FUNCTION_BLOCK PearlingHdl

(*
	Description 	: Function bloc to handle pearling unit
	Author		: DLA
	Date		: 09.06.2014
	Version		: 1.00

	Modifications :
                                                                                                                                                                                 
*)

VAR_INPUT
	bEnable									: BOOL;										// Not used
	bPowerOn								: BOOL;										// Power activate
	eCommand								: TModuleCommands;							// Module commande
	bHomeX									: BOOL;										// Axe X Sensor home
	bLimitPosX								: BOOL;										// Axe X Sensor positif limite position
	bLimitNegX								: BOOL;										// Axe X Sensor negatif limite position
	bHomeY									: BOOL;										// Axe Y Sensor home
	bLimitPosY								: BOOL;										// Axe Y Sensor positif limite position 
	bLimitNegY								: BOOL;										// Axe Y Sensor negatif limite position 
	bHomeZ1									: BOOL;										// Axe Z1 Sensor home
	bLimitPosZ1								: BOOL;										// Axe Z1 Sensor positif limite position
	bLimitNegZ1								: BOOL;										// Axe Z1 Sensor negatif limite position
	bHomeZ2									: BOOL;										// Axe Z2 Sensor home
	bLimitPosZ2								: BOOL;										// Axe Z2 Sensor positif limite position
	bLimitNegZ2								: BOOL;										// Axe Z2 Sensor negatif limite position
	bChuck1Opened							: BOOL;										// Chuck Z1 is opened
	bChuck1Closed							: BOOL;										// Chuck Z1 is closed
	bChuck2Opened							: BOOL;										// Chuck Z2 is opened
	bChuck2Closed							: BOOL;										// Chuck Z2 is closed
	bResetErrors							: BOOL;										// Reseting the errors on the module
	bNewJob									: BOOL;										// New job loaded
	bStopReq								: BOOL;										// Request for stoping the module
	bPauseReq								: BOOL;										// Request for pausing the module
	asStickData								: ARRAY[0..1] OF TStickData;				// Description of the sticks used
	asStickDataMMI							: ARRAY[0..1] OF TStickDataMMI;				// Information for the use of the sticks from HMI
	sStickDataShared						: TStickDataShared;							// Information shared betweeen modules for the use of the sticks from HMI
	lrCompenseWeight1						: LREAL;									// Z1 weight compensation
	lrCompenseWeight2						: LREAL;									// Z2 weight compensation
	iComPort								: INT;										// 
	sInTakeFromBarrel						:TGiver;
	iContact1Distance						: INT;
	iContact2Distance						: INT;
	iLoadSensorValue						: INT;
	eSharpenRunStatus						: TRunStatus;
	eBarrelRunStatus						: TRunStatus;
	eRunCommand								: TRunCmdPearling;
	bKeepBothHeadWarm						: BOOL;
	eTableSideForLoader						: TTableSide;
	sPartData								: TPartDataMMI;
	bHead1IsUsed							: BOOL;
	bHead2IsUsed							: BOOL;
	bParallelProduction						: BOOL;
	iLeftVacuumFlow							: INT;
	iRightVacuumFlow						: INT;
	iMachineWO								: DINT;
	iMachineSN								: INT;
	yModulePosition							: BYTE;
END_VAR
VAR_OUTPUT
	bModuleError							: BOOL;
	bXAxisError								: BOOL;
	bYAxisError								: BOOL;
	bZ1AxisError							: BOOL;
	bZ2AxisError							: BOOL;
	bChuck1Error							: BOOL;
	bChuck2Error							: BOOL;
	bSpindle1Error							: BOOL;
	bSpindle2Error							: BOOL;
	bSecurityError							: BOOL;
	bSecurityErrorDetected					: BOOL;
	bMCRError								: BOOL;
	bStick1Broken							: BOOL;
	bStick2Broken							: BOOL;
	bStartPearlingMotor1					: BOOL;
	bStartPearlingMotor2					: BOOL;
	bOpenChuck1								: BOOL;
	bOpenChuck2								: BOOL;
	bActivateEject1							: BOOL;
	bActivateEject2							: BOOL;
	bActivateBlowing1						: BOOL;
	bActivateBlowing2						: BOOL;
	bAspirationPearling1On					: BOOL;
	bAspirationPearling2On					: BOOL;
	bAspirationSharpenOn					: BOOL;
	bStickContact1							: BOOL;
	bStickContact2							: BOOL;
	bCurrent1ReadError						: BOOL;
	bCurrent2ReadError						: BOOL;
	bMotor1Error							: BOOL;
	bMotor2Error							: BOOL;
	bPearlingWeight1OutOfToleranceError		: BOOL;
	bPearlingWeight2OutOfToleranceError		: BOOL;
	bStickNotTakenError						: BOOL;
	bReady2ChangeTool						: BOOL;
	iStickHead								: INT;
	sOutTakeFromBarrel						: TTaker;
	eSharpenRunCmd							: TRunCmdSharpen;
	eBarrelRunCmd							: TRunCmdBarrel;
	eRunStatus								: TRunStatus;
	bManInterlockOut						: BOOL;
	adwMotorRunningHours					: ARRAY[0..1] OF DWORD;
	adwSpindleRunningHours					: ARRAY[0..1] OF DWORD;
	bLeftSpindleUsedWarning					: BOOL;
	bRightSpindleUsedWarning				: BOOL;
	bLeftMotorUsedWarning					: BOOL;
	bRightMotorUsedWarning					: BOOL;
	bLeftSpindleLimitWarning				: BOOL;
	bRightSpindleLimitWarning				: BOOL;
	bLeftSpindleHeatWarning					: BOOL;
	bRightSpindleHeatWarning				: BOOL;
END_VAR
VAR_IN_OUT
	sCurrentState							: TModuleData;
	TManualCmd								: TManPearling;
	sRecData								: ComBuffer;
	sTransData								: ComBuffer;
	asPearlData								: ARRAY[0..1] OF TMMIPearlData;
	sXAxisRef								: AXIS_REF;
	sYAxisRef								: AXIS_REF;
	sZ1AxisRef								: AXIS_REF;
	sZ2AxisRef								: AXIS_REF;
	sRunData								: TRunDataPearling;
	asProbingLog							: ARRAY[0..1] OF  TProbingLog;
END_VAR
VAR PERSISTENT
	alrHighDynParams						: ARRAY[0..3] OF TDynAxisParam;
	alrLowDynParams							: ARRAY[0..3] OF TDynAxisParam;
	alrSafePos								: ARRAY[0..3] OF LREAL;
	alrRobotPos								: ARRAY[0..3,0..PTP_END] OF LREAL;					(* XYZ1Z2 for Ref/Inner/Outer/Drop/... *)
	alrJogStep								: ARRAY[0..3] OF LREAL;								(* Jog step for X,Y,Z1,Z2 *)
	lrSharpeningDelta						: LREAL								:= 10;
	lrSharpenPosOffset						: LREAL								:= 2;
	alrChuckRetractOffset					: ARRAY[0..1] OF LREAL				:= [1,1];		// TODO: HFO, modifier valeur, original [2, 2]
	lrStickTakeSpeed						: LREAL								:= 10;
	bBypassMCR								: BOOL;
(*	iMaxNbOfFwBwSharpen						: INT	:= 1;*)
	TBreakStickDetectTime					: TIME	:= t#30ms;
	aiContactThresholdArea					: ARRAY[0..1, 0..PA_END] OF INT;
	aiSpindleManualSpeed					: ARRAY[0..1] OF INT;
	alrSensorRate							: ARRAY[0..1] OF LREAL								(* in Unit / mm *);
	lrSensorZSpeed							: LREAL								:= 0.1;
	alrLoadSensorOffset						: ARRAY[0..1] OF LREAL;
	lrLoadSensorRate						: LREAL								:= 6.36121;			(* in Unit / g *)
	iLoadSensorTare							: INT								:= 3175;		(* in Unit / g *)
	alrRatiog2mm							: ARRAY[0..1] OF LREAL				:= [2(0.001)];
	lrStickErrorDeltaPos					: LREAL								:= 0.5;
(*	lrSpindelOffsetX						: LREAL								:= 50.0;*)
	iMCROffsetCurrent						: ARRAY[0..1] OF INT				:= [0,0];
	iMCRCurrentRatio						: ARRAY[0..1] OF INT				:= [1,1];
	aiMotorStartedTimeout					: ARRAY[0..1] OF INT 				:= [2000,2000]; (* in ms *)
	aiMotorStoppedTimeout					: ARRAY[0..1] OF INT 				:= [2000,2000]; (* in ms *)
	bForceProbing							: BOOL;
	lrStickOutAfterChange					: LREAL 							:= 12; 			(* mm *)
	lrProbingThreshold						: LREAL								:= 0.05; 		(* mm *)
	alrSharpenTeachZOffset					: LREAL								:= 0.4;
	dwMaxSpindleRunningHours				: DWORD								:= 900;			(*Hours : Max time running spindle before changing it *)
	dwMaxMotorRunningHours					: DWORD								:= 2000;		(*Hours : Max time running motor before changing it *)
	iMCRMinThCurrent						: INT								:= 200;
	iMCRMaxThCurrent 						: INT								:= 800;
	iMCRWarnThCurrent 						: INT								:= 600;
	adwPearlsCounter 						: ARRAY[0..1] OF DWORD				:= [2(0)];
	lrCenterSharpningOffset 				: LREAL 							:= 1.5;
	lrSecurityPreRefPosZ					: LREAL 							:= 1.5;
END_VAR
VAR CONSTANT
	lrLoadSensorStep						: LREAL								:= 0.02;
	lrWeightCalibrationStartOffsetZ			: LREAL 							:= 0.1;
	lrSafeTolerance 						: LREAL 							:= 1;			(* Tolerance for safety Z axis down *)
	lrMaxXYMoveAllowed						: LREAL 							:= 30;			(* Max move authorized when Z axis is down *)
	lrManMaxXYMoveAllowed					: LREAL 							:= 2.1;			(* Max move in manual mode authorized when Z axis is down *)
	lrSecurityRadius						: LREAL								:= 18;
	bInvertX								: BOOL 								:= FALSE;
	bInvertY								: BOOL 								:= FALSE;
	bInvertZ								: BOOL 								:= TRUE;
	lrLayeringCenterOffsetXTable			: LREAL 							:= 65;
	lrLayeringCenterOffsetYTable			: LREAL 							:= 18;
	iHeatOnSpeed							: INT								:= 1000;
END_VAR
VAR
	alrMaxRobotSpeed						: ARRAY[0..3] OF LREAL;
	alrManualRobotSpeed						: ARRAY[0..3] OF LREAL;
	i										: INT;
	j										: INT;
	iAxis									: INT;
	iCurrentManAxis							: INT;
	eRobotXYStatus							: TAxisState;
	aeMoveRobotCommand						: ARRAY[0..3] OF TAxisCommands		:= [4(AC_None)];
	aTRobotAxis								: ARRAY[0..3] OF StdAxis;
	alrCurrentSpeed							: ARRAY[0..3] OF LREAL;
	alrTargetPos							: ARRAY[0..3] OF LREAL;
(*	abForceNewPosZ							: ARRAY[0..1] OF BOOL;*)
	nPearlIndex								: UINT;
	aTPearlingTimer							: ARRAY[0..1] OF TON;
	TCheckTimer								: TON;
	alrPreRefPosZ							: ARRAY[0..1] OF LREAL;
(*	bRemoveXLimitSecurity					: BOOL;
	bRemoveYLimitSecurity					: BOOL;*)
	bManualZIsSafe							: BOOL;
	abChangeStick							: ARRAY[0..1] OF BOOL				:= [TRUE,TRUE];
	abSharpenStick							: ARRAY[0..1] OF BOOL				:= [TRUE,TRUE];
	abDoProbing								: ARRAY[0..1] OF BOOL;
	abRetryProbing							: ARRAY[0..1] OF BOOL;
	abProbingDone							: ARRAY[0..1] OF BOOL;
	aiProbingCount							: ARRAY[0..1] OF INT;
	alrProbingStartPos						: ARRAY[0..1] OF LREAL;
	eStickStep								: TModuleSteps;
	aeProbingStep							: ARRAY[0..1] OF TModuleSteps;
	TCheckTime								: TIME								:= T#5S;
	TMCRDrv									: MCRDrv;
	aTCheckChuck							: ARRAY[0..1] OF FB_CheckJack1_2;
	alrCorrectionMCR						: ARRAY[0..1] OF LREAL;
	eMCRCommand								: TMCRCommands;
	bMCRReady								: BOOL;
(*	abLastStickContact						: ARRAY[0..1] OF BOOL;*)
	aiNbOfPearlsDone						: ARRAY[0..1] OF INT;
	iCurrentArea							: INT;
	aArea									: ARRAY[0..C_MAX_NB_OF_PEARLS] OF TPearlsArea;
	alrPearlingEnergy						: ARRAY[0..1] OF LREAL;
	aTDispersion							: ARRAY[0..1] OF Dispersion;
	alrRemainingStickLength					: ARRAY[0..1] OF LREAL;
	aTMotorCounter							: ARRAY[0..1] OF RunningCounter;
	aTSpindleCounter						: ARRAY[0..1] OF RunningCounter;
	TWaitChuckOpen							: TON;
	abZRefTaken								: ARRAY[0..3,0..1,0..1] OF BOOL; 					(*Layring , Offset Layring, Head *)
	alrSecurityPosition						: ARRAY[0..3,0..1,0..1] OF LREAL;					(*Layring , Offset Layring, Head *)
	alrContactPosition						: ARRAY[0..3,0..1,0..1] OF LREAL;					(*Layring , Offset Layring, Head *)
	alrContactStickPosition					: ARRAY[0..3,0..1,0..1] OF LREAL;					(*Layring , Offset Layring, Head *)
	alrProbingRef							: ARRAY[0..3,0..1,0..1] OF LREAL; 					(*Layring , Offset Layring, Head *)
	alrHeadSecurityPosition					: ARRAY[0..1] OF LREAL;
	alrHeadContactPosition					: ARRAY[0..1] OF LREAL;
	alrHeadContactStickPosition				: ARRAY[0..1] OF LREAL;
	alrHeadProbingRef						: ARRAY[0..1] OF LREAL;
	alrSharpenProbing						: ARRAY[0..1] OF LREAL;
	alrDeltaSharpenProbing					: ARRAY[0..1] OF LREAL;
	alrStickCorrection						: ARRAY[0..1] OF LREAL;
	alrDeltaStickCorrection					: ARRAY[0..1] OF LREAL;
	alrFirstPearlCorrection					: ARRAY[0..1] OF LREAL;
	abTakeZRef								: ARRAY[0..1] OF BOOL;
	bClearZRef								: BOOL;
	abNeedSharpening						: ARRAY[0..1] OF BOOL;
	abNeedChangeStick						: ARRAY[0..1] OF BOOL;
	bFirstStart								: BOOL								:= TRUE;
	bFirstInit								: BOOL								:= TRUE;
	abBadPearling							: ARRAY[0..1] OF BOOL;
	alrDynParams							: ARRAY[0..3] OF TDynAxisParam;
	yMCRChannel								: BYTE;
	abPearlStarted							: ARRAY[0..1] OF BOOL;
	abPearlDone								: ARRAY[0..1] OF BOOL;
	abPearlPosReached						:  ARRAY[0..1] OF BOOL;
	lrRadius								: LREAL;
	alrLastProbingPos						: ARRAY[0..1] OF LREAL;
	aTWaitMotorStarted						: ARRAY[0..1] OF TON;
	aTWaitMotorStopped						: ARRAY[0..1] OF TON;
	iNbOfFwBwSharpen						: INT;
	iNbOfFwBwSharpenBeforeMove				: INT;
	abNewStick								: ARRAY[0..1] OF BOOL				:= [FALSE,FALSE];
	iDebugPos								: INT;
	iDebugSide								: INT;
	aTDetectStickBroken						: ARRAY[0..1] OF TON;
(*	bZIsSafe								: BOOL;*)
	alrProbingPos							: ARRAY[0..1] OF LREAL;
	alrCheckProbingPos						: ARRAY[0..1] OF LREAL;
	alrProbingLimit							: ARRAY[0..1] OF LREAL;
(*	iNbOfPearlsRemainingOnThisArea			: INT;*)
	abCheckingStick							: ARRAY[0..1] OF BOOL;
	TWaitCurrentMotorBeltOk					: TON;
	TWaitCurrentMotorWarmOk					: TON;
	aTStickContactValidated					: ARRAY[0..1] OF TON;
	TStickContactValidTime					: TIME								:= T#250MS; // valeur original ==> t#500ms; Temps de stabilisation du capteur de de distance en contacte
	TStickStabilisationTime					: TIME								:= T#400MS;	// Temps pour stabiliser le capteur de distance sans contact
	aIMinPos								: ARRAY[0..1] OF INT;
	alrDeltaZPearl							: ARRAY[0..1] OF LREAL;
	alrDeltaWeightPearl						: ARRAY[0..1] OF LREAL;
	iTableIndex								: INT;
	lrBasePos								: LREAL;
(*	TWaitEjectorTimer						: TON;*)
	abWeightTableValid						: ARRAY[0..1] OF BOOL;
	alrWeightTable							: ARRAY[0..1,0..C_WEIGHT_TABLE_MAX] OF LREAL;
	iSide									: INT;
	abStartPearlingMotor					: ARRAY[0..1] OF BOOL;
	aiContactDistance						: ARRAY[0..1] OF INT;
	abUseSpindle							: ARRAY[0..1] OF BOOL;
	abChuckOpened							: ARRAY[0..1] OF BOOL;
	abChuckClosed							: ARRAY[0..1] OF BOOL;
	abOpenChuck								: ARRAY[0..1] OF BOOL;
	abActivateEject							: ARRAY[0..1] OF BOOL;
	abSpindleError							: ARRAY[0..1] OF BOOL;
	abAspirationPearling					: ARRAY[0..1] OF BOOL;
	abStickContact							: ARRAY[0..1] OF BOOL;
	abActivateBlowing						: ARRAY[0..1] OF BOOL;
	abCurrentReadError						: ARRAY[0..1] OF BOOL;
	abMotorError							: ARRAY[0..1] OF BOOL;
	abSpindleCurrentOk						: ARRAY[0..1] OF BOOL;
	abStickBroken							: ARRAY[0..1] OF BOOL;
	abStickBrokenDetected					: ARRAY[0..1] OF BOOL;
	abPearlNeeded							: ARRAY[0..1] OF BOOL;
	abHeadIsUsed							: ARRAY[0..1] OF BOOL;
	abPearlingWeightOutOfToleranceError		: ARRAY[0..1] OF BOOL;
	abPearlingWeightOutOfToleranceDetected	: ARRAY[0..1] OF BOOL;
	abFirstPearl							: ARRAY[0..1] OF BOOL;
	aiCountPearlError						: ARRAY[0..1] OF INT;
	alrBasePearlingEnergy					: ARRAY[0..1] OF LREAL;
	alrCompenseWeight						: ARRAY[0..1] OF LREAL;
	aiPearlingLayringPos					: ARRAY[0..1] OF INT;
	aiPearlingLayringOffsetPos				: ARRAY[0..1] OF INT;
	anPearlIndexDone						: ARRAY[0..1] OF UINT;
	aiSideInfo								: ARRAY[0..1] OF INT;
	TLayeringCenter							:  TPositionXY;
	TPearlPosition							:  TPositionXY;
	iFirstHeadUsed							: INT;
	iRejectPos								: INT;
	iChangeStickPos							: INT;
	nPearl									: UINT;
	aiPearlingTeachedPos					: ARRAY[0..1] OF INT;
	alrPearlingOffset						: ARRAY[0..4] OF LREAL;
	alrPearlingInvert						: ARRAY[0..4] OF LREAL;
	alrHeadPushed_mm						: ARRAY[0..1] OF LREAL;
(*	psPartData								: ARRAY[0..1] OF POINTER TO TPartData;*)
	bChangeToolSide							: BOOL;
(*	bChangeTool								: BOOL;*)
	bEndPearling							: BOOL;
	lrWeight								: LREAL;
	lrMaxMCRCorrection						: LREAL;
	bCalibrationInProgress					: BOOL;
	aeProbingArea							: ARRAY[0..1] OF TProbingArea;
	TDebug									: TPearlingDebug;
	aePearlingArea							: ARRAY[0..1] OF TProbingArea;
	TWaitHeadStab							: TON;
	atStickValidateTime						: ARRAY[0..1] OF LREAL;
	aiVacuumFlow							: ARRAY[0..1] OF INT;
	ayChannelStatus							: ARRAY[0..1] OF BYTE;
	abCurrentLimitWarning					: ARRAY[0..1] OF BOOL;
	aTWaitSpindleHeatOn						: ARRAY[0..1] OF TON;
	aTDetectSpindleCooled					: ARRAY[0..1] OF TON;
	abNeedSpindleHeatOn						: ARRAY[0..1] OF BOOL;
	ai_ProbingStep							: ARRAY [0..1] OF INT;
	i_StickStep								: INT;
	iDebugPosBrokenStick					: INT;
END_VAR


(*_AppInfo.BootDataLoaded;			// HFO, to know if boot data was loaded
_AppInfo.OldBootData;
_AppInfo.PersistentStatus;*)

(* Optimize code *)
abStartPearlingMotor[PH_Left] := bStartPearlingMotor1;
abStartPearlingMotor[PH_Right] := bStartPearlingMotor2;
aiContactDistance[PH_Left] := iContact1Distance;
aiContactDistance[PH_Right] := iContact2Distance;
abChuckOpened[PH_Left] := bChuck1Opened;
abChuckOpened[PH_Right] := bChuck2Opened;
abChuckClosed[PH_Left] := bChuck1Closed;
abChuckClosed[PH_Right] := bChuck2Closed;
alrCompenseWeight[PH_Left] := lrCompenseWeight1;
alrCompenseWeight[PH_Right] := lrCompenseWeight2;
abHeadIsUsed[PH_Left] := bHead1IsUsed;
abHeadIsUsed[PH_Right] := bHead2IsUsed;
aiVacuumFlow[PH_LEFT] := iLeftVacuumFlow;
aiVacuumFlow[PH_RIGHT] := iRightVacuumFlow;

eSharpenRunCmd := RCS_None;
eBarrelRunCmd := RCB_None;

IF bInvertX THEN
	alrPearlingInvert[PA_X] := -1;
ELSE
	alrPearlingInvert[PA_X] := 1;
END_IF
IF bInvertY THEN
	alrPearlingInvert[PA_Y] := -1;
ELSE
	alrPearlingInvert[PA_Y] := 1;
END_IF
IF bInvertZ THEN
	alrPearlingInvert[PA_Z1] := -1;
	alrPearlingInvert[PA_Z2] := -1;
ELSE
	alrPearlingInvert[PA_Z1] := 1;
	alrPearlingInvert[PA_Z2] := 1;
END_IF

FOR iAxis := 0 TO 3 DO
	alrMaxRobotSpeed[iAxis] := aTRobotAxis[iAxis].lrRunningSpeed;
	alrManualRobotSpeed[iAxis] := aTRobotAxis[iAxis].lrManualSpeed;
END_FOR

IF (NOT sCurrentState.bStepMode) THEN
	sCurrentState.bWaitStep := FALSE;
END_IF

IF bFirstStart THEN
	FOR iSide := 0 TO 1 DO
		abWeightTableValid[iSide] := FALSE;
		aTDetectSpindleCooled[iSide](IN := FALSE);
		aTWaitSpindleHeatOn[iSide](IN := FALSE);
		abNeedSpindleHeatOn[iSide] := TRUE;
	END_FOR
	bFirstStart := FALSE;
END_IF

IF bNewJob THEN
	FOR iSide := 0 TO 1 DO
		abSharpenStick[iSide] := TRUE;
		aiNbOfPearlsDone[iSide] := 1;
	END_FOR
	bClearZRef := TRUE;
END_IF

FOR iSide:=0 TO 1 DO
	abStickContact[iSide] := aiContactDistance[iSide] > (aiContactThresholdArea[iSide , aeProbingArea[iSide]] + 0.05 * alrSensorRate[iSide]);
	aTWaitMotorStarted[iSide](IN := abStartPearlingMotor[iSide],PT := INT_TO_TIME(aiMotorStartedTimeout[iSide]));
	aTWaitMotorStopped[iSide](IN := NOT abStartPearlingMotor[iSide],PT := INT_TO_TIME(aiMotorStoppedTimeout[iSide]));
	aTMotorCounter[iSide](bStart := abStartPearlingMotor[iSide], bReset := FALSE);
	aTSpindleCounter[iSide](bStart := abStartPearlingMotor[iSide], bReset := FALSE);
	IF NOT abDoProbing[iSide] THEN
		abProbingDone[iSide] := FALSE;
	END_IF
	(* For debug purpose *)
	IF alrSensorRate[iSide] <> 0 THEN
		alrHeadPushed_mm[iSide] := INT_TO_REAL(LREAL_TO_INT(((aiContactDistance[iSide]-aiContactThresholdArea[iSide , aeProbingArea[iSide]])/alrSensorRate[iSide])*100))/100.0;
	ELSE
		alrHeadPushed_mm[iSide] := 0;
	END_IF
	alrBasePearlingEnergy[iSide] := sRunData.sPearlingData.iWeight +  alrCompenseWeight[iSide];
	IF bParallelProduction THEN
		aiSideInfo[iSide] := 0;
	ELSE
		aiSideInfo[iSide] := iSide;
	END_IF
END_FOR

(* For debug purpose *)
IF lrLoadSensorRate<>0 THEN
	lrWeight := (INT_TO_LREAL(iLoadSensorValue) - INT_TO_LREAL(iLoadSensorTare)) / lrLoadSensorRate;
ELSE
	lrWeight := 0;
END_IF

CASE eCommand OF
	MC_NoCmd :
		CASE sCurrentState.eStatus OF
			MS_Init :
				CASE sCurrentState.eStep OF
(*----------------- Init ------------------*)
					SP_InitStp1 :
						FOR iSide := 0 TO 1 DO
							abAspirationPearling[iSide] := FALSE;
							abActivateEject[iSide] := FALSE;
							(* Move Z Up *)
							aeMoveRobotCommand[PA_Z1+iSide] := AC_MoveLimitNeg;
						END_FOR
						bAspirationSharpenOn := FALSE;
						alrCurrentSpeed := alrMaxRobotSpeed;
						sCurrentState.eStep := SP_InitStp2;
					SP_InitStp2 :
						IF aTRobotAxis[PA_Z1].eCurrentState = AS_OnLimitNeg  AND
						     aTRobotAxis[PA_Z2].eCurrentState = AS_OnLimitNeg THEN
							(* Init X / Y*)
							aeMoveRobotCommand[PA_X] := AC_Init;
							aeMoveRobotCommand[PA_Y] := AC_Init;
							sCurrentState.eStep := SP_InitStp3;
						END_IF
					SP_InitStp3 :
						IF 	(aTRobotAxis[PA_X].eCurrentState = AS_InPosition) AND
							(aTRobotAxis[PA_Y].eCurrentState = AS_InPosition) THEN
							(* Move X/ Y to Safe *)
							alrTargetPos[PA_X] := alrSafePos[PA_X];
							alrTargetPos[PA_Y] := alrSafePos[LA_Y];
							aeMoveRobotCommand[PA_X] := AC_MoveAtAbsPos;
							aeMoveRobotCommand[PA_Y] := AC_MoveAtAbsPos;
							sCurrentState.eStep := SP_InitStp4;
						END_IF
					SP_InitStp4 :
						IF aTRobotAxis[PA_X].eCurrentState = AS_InPosition AND
						     aTRobotAxis[PA_Y].eCurrentState = AS_InPosition THEN
								(* Init Z *)
								aeMoveRobotCommand[PA_Z1] := AC_Init;
								aeMoveRobotCommand[PA_Z2] := AC_Init;
								sCurrentState.eStep := SP_InitStp5;
						END_IF
					SP_InitStp5 :
						IF aTRobotAxis[PA_Z1].eCurrentState=AS_InPosition AND
							aTRobotAxis[PA_Z2].eCurrentState=AS_InPosition THEN
							(* Move Z to Safe *)
							alrTargetPos[PA_Z1] := alrSafePos[PA_Z1];
							alrTargetPos[PA_Z2] := alrSafePos[LA_Z2];
							aeMoveRobotCommand[PA_Z1] := AC_MoveAtAbsPos;
							aeMoveRobotCommand[PA_Z2] := AC_MoveAtAbsPos;
							sCurrentState.eStep := SP_InitStp6;
						END_IF
					SP_InitStp6 :
						IF  aTRobotAxis[PA_Z1].eCurrentState = AS_InPosition AND
						     aTRobotAxis[PA_Z2].eCurrentState = AS_InPosition THEN
							IF bBypassMCR THEN
								sCurrentState.eStep := SP_InitStp99;
							ELSIF bMCRReady THEN
								yMCRChannel := 1;
								sCurrentState.eStep := SP_InitStp10;
							END_IF
						END_IF
					SP_InitStp10 :
						(* Configure MCR *)
						eMCRCommand := MCRC_ConfigMeasure;
						sCurrentState.eStep := SP_InitStp11;
					SP_InitStp11 :
						IF bMCRReady THEN
							IF yMCRChannel = 1 THEN
								yMCRChannel := 2;
								sCurrentState.eStep := SP_InitStp10;
							ELSE
								yMCRChannel := 1;
								sCurrentState.eStep := SP_InitStp12;
							END_IF
						END_IF
					SP_InitStp12 :
						eMCRCommand := MCRC_SetRatio;
						TMCRDrv.lrRatio := asStickDataMMI[yMCRChannel - 1].lrMCRRatio;
						sCurrentState.eStep := SP_InitStp13;
					SP_InitStp13 :
						IF bMCRReady THEN
							IF yMCRChannel = 1 THEN
								yMCRChannel := 2;
								sCurrentState.eStep := SP_InitStp12;
							ELSE
								yMCRChannel := 1;
								sCurrentState.eStep := SP_InitStp14;
							END_IF
						END_IF
					SP_InitStp14 :
						(* Do spindle heat on if needed *)
						TMCRDrv.iSpeedSetpoint := iHeatOnSpeed;;
						eMCRCommand := MCRC_SetSpeed;
						sCurrentState.eStep := SP_InitStp15;
					SP_InitStp15 :
						IF bMCRReady THEN
							IF yMCRChannel = 1 THEN
								yMCRChannel := 2;
								sCurrentState.eStep := SP_InitStp14;
							ELSE
								yMCRChannel := 1;
								sCurrentState.eStep := SP_InitStp16;
							END_IF
						END_IF
					SP_InitStp16 :
						abStartPearlingMotor[PH_Left] := abNeedSpindleHeatOn[PH_Left];
						abStartPearlingMotor[PH_Right] := abNeedSpindleHeatOn[PH_Right];
						sCurrentState.eStep := SP_InitStp17;
					SP_InitStp17 :
						IF (NOT (abNeedSpindleHeatOn[PH_Left] AND abStartPearlingMotor[PH_Left]) AND 
								NOT (abNeedSpindleHeatOn[PH_Right] AND abStartPearlingMotor[PH_Right])) THEN
							sCurrentState.eStep := SP_InitStp25;
						END_IF
					SP_InitStp25 :
						eMCRCommand := MCRC_SetSpeed;
						TMCRDrv.iSpeedSetpoint := sStickDataShared.sStickDataMMIShared.iMCRSharpenSpeed;
						sCurrentState.eStep := SP_InitStp26;
					SP_InitStp26 :
						IF bMCRReady THEN
							IF yMCRChannel = 1 THEN
								yMCRChannel := 2;
								sCurrentState.eStep := SP_InitStp25;
							ELSE
								yMCRChannel := 1;
								sCurrentState.eStep := SP_InitStp27;
							END_IF
						END_IF
					SP_InitStp27:
						(* Set Parameter*)
						IF NOT bFirstInit THEN
							eMCRCommand := MCRC_SetParam;
							TMCRDrv.iOffsetCurrent := iMCROffsetCurrent[yMCRChannel - 1];
							TMCRDrv.iCurrentRatio := iMCRCurrentRatio[yMCRChannel - 1];
						END_IF
						sCurrentState.eStep := SP_InitStp28;
					SP_InitStp28:
						IF bMCRReady THEN
							IF yMCRChannel = 1 THEN
								yMCRChannel := 2;
								sCurrentState.eStep := SP_InitStp27;
							ELSE
								yMCRChannel := 1;
								sCurrentState.eStep := SP_InitStp29;
							END_IF
						END_IF
					SP_InitStp29:
						(* Set threshold*)
						eMCRCommand := MCRC_DefineCurrentThr;
						TMCRDrv.iMinThCurrent := iMCRMinThCurrent;
						TMCRDrv.iMaxThCurrent := iMCRMaxThCurrent;
						TMCRDrv.iWarnThCurrent := iMCRWarnThCurrent;
						sCurrentState.eStep := SP_InitStp30;
					SP_InitStp30:
						IF bMCRReady THEN
							IF yMCRChannel = 1 THEN
								yMCRChannel := 2;
								sCurrentState.eStep := SP_InitStp29;
							ELSE
								yMCRChannel := 1;
								sCurrentState.eStep := SP_InitStp31;
							END_IF
						END_IF
					SP_InitStp31:
						IF NOT bFirstInit THEN
							(* Set MachineID*)
							eMCRCommand := MCRC_DefineMachineID;
							TMCRDrv.iMachineWO := iMachineWO;
							TMCRDrv.iMachineSN := iMachineSN;
							TMCRDrv.yMachineSide := asc('a') + yModulePosition;
						END_IF
						sCurrentState.eStep := SP_InitStp32;
					SP_InitStp32:
						IF bMCRReady THEN
							IF yMCRChannel = 1 THEN
								yMCRChannel := 2;
								sCurrentState.eStep := SP_InitStp31;
							ELSE
								yMCRChannel := 1;
								sCurrentState.eStep := SP_InitStp99;
							END_IF
						END_IF
					SP_InitStp50: (*Init if already init done, always move Z to safe *)
						(* Go to safe position *)
						alrCurrentSpeed := alrMaxRobotSpeed;
						alrTargetPos[PA_Z1] := alrSafePos[PA_Z1];
						alrTargetPos[PA_Z2] := alrSafePos[PA_Z2];
						aeMoveRobotCommand[PA_Z1] := AC_MoveAtAbsPos;
						aeMoveRobotCommand[PA_Z2] := AC_MoveAtAbsPos;
						sCurrentState.eStep := SP_InitStp51;
					SP_InitStp51 :
						IF 	(aTRobotAxis[PA_Z1].eCurrentState = AS_InPosition) AND
							(aTRobotAxis[PA_Z2].eCurrentState = AS_InPosition) THEN
							sCurrentState.eStep := SP_InitStp99;
						END_IF
					SP_InitStp99 :
						bFirstInit := FALSE;
						FOR iSide := 0 TO 1 DO
							abDoProbing[iSide] := FALSE;
							abUseSpindle[iSide] := FALSE;
							abRetryProbing[iSide] := FALSE;
							aiProbingCount[iSide] := 0;
						END_FOR
						sCurrentState.eStatus := MS_Ready;
						sCurrentState.bInitDone := TRUE;
						sCurrentState.eStep := SP_RunStp1;
						eStickStep := SP_RunStp1;
						aeProbingStep[PH_Left] := SP_RunStp1;
						aeProbingStep[PH_Right] := SP_RunStp1;

				END_CASE
			MS_Running :
				IF (NOT sCurrentState.bWaitStep) THEN
(*----------------- Probing ------------------*)
					FOR iSide := 0 TO 1 DO
						CASE aeProbingStep[iSide] OF
							SP_RunStp1 :
								IF abDoProbing[iSide] THEN
									aiProbingCount[iSide] := 0;
									alrProbingStartPos[iSide] := alrTargetPos[PA_Z1 + iSide];
									abProbingDone[iSide] := FALSE;
									abStartPearlingMotor[iSide] := FALSE;
									aeProbingStep[iSide] := SP_RunStp20;
								END_IF
							SP_RunStp20:
								(* Continuous move probing with analog sensor *)
								IF (aTRobotAxis[PA_Z1+ iSide].eCurrentState = AS_InPosition) AND aTWaitMotorStopped[iSide].Q THEN
									(* Move 0.5 mm above probing pos to check default sensor value *)
									alrTargetPos[PA_Z1 + iSide] := alrProbingStartPos[iSide] - 0.5;		// TODO : HFO modifier valeur en dure, original 0.5
									alrCurrentSpeed[PA_Z1 + iSide] := alrMaxRobotSpeed[PA_Z1 + iSide];
									aeMoveRobotCommand[PA_Z1 + iSide] := AC_MoveAtAbsPos;
									aTStickContactValidated[iSide](IN := FALSE);
									aeProbingStep[iSide] := SP_RunStp21;
								END_IF
							SP_RunStp21:
								IF (aTRobotAxis[PA_Z1 + iSide].eCurrentState = AS_InPosition) THEN
									aTStickContactValidated[iSide](IN := TRUE,PT := TStickStabilisationTime);	// Valueur original ==> PT := TStickContactValidTime
									IF aTStickContactValidated[iSide].Q THEN
										asProbingLog[iSide].iPreviousProbingThreshold := aiContactThresholdArea[iSide , aeProbingArea[iSide]];
										aiContactThresholdArea[iSide , aeProbingArea[iSide]] := aiContactDistance[iSide];
										(* Move down 0.5mm *)
										alrTargetPos[PA_Z1 + iSide] := alrProbingStartPos[iSide]- 0.3;  		// TODO : HFO, Ajout de valeur negative
										//alrTargetPos[PA_Z1 + iSide] := alrProbingStartPos[iSide];
										aeMoveRobotCommand[PA_Z1 + iSide] := AC_MoveAtAbsPos;
										aTStickContactValidated[iSide](IN := FALSE);
										aeProbingStep[iSide] := SP_RunStp25;
									END_IF
								END_IF
							SP_RunStp25:
								IF (aTRobotAxis[PA_Z1 + iSide].eCurrentState = AS_InPosition) THEN
									aTStickContactValidated[iSide](IN := TRUE,PT := TStickContactValidTime);
									IF aTStickContactValidated[iSide].Q THEN
										(* Check if we must go up or down *)
										IF (aiContactDistance[iSide] > aiContactThresholdArea[iSide , aeProbingArea[iSide]] + alrSensorRate[iSide] * lrProbingThreshold) THEN
											(* Go up *)
											aeProbingStep[iSide] := SP_RunStp30;
										ELSE
											(* Go down *)
											aeProbingStep[iSide] := SP_RunStp40;
										END_IF								
									END_IF
								END_IF	
							SP_RunStp30:
								(* Move up slowly until we get contact *)
								alrTargetPos[PA_Z1 + iSide] := alrProbingStartPos[iSide] - 2;
								alrCurrentSpeed[PA_Z1 + iSide] := lrSensorZSpeed;
								aeMoveRobotCommand[PA_Z1 + iSide] := AC_MoveAtAbsPos;
								aeProbingStep[iSide] := SP_RunStp35;
							SP_RunStp35:
								IF (aiContactDistance[iSide] < aiContactThresholdArea[iSide , aeProbingArea[iSide]] + alrSensorRate[iSide] * lrProbingThreshold) THEN
									aTStickContactValidated[iSide](IN := FALSE);
									aeMoveRobotCommand[PA_Z1 + iSide] := AC_Stop;
									aeProbingStep[iSide] := SP_RunStp50;
									sCurrentState.bWaitStep := TRUE;
								ELSIF (aTRobotAxis[PA_Z1 + iSide].eCurrentState = AS_InPosition) THEN
									aeMoveRobotCommand[PA_Z1] := AC_Stop;
									aeMoveRobotCommand[PA_Z2] := AC_Stop;
									bSecurityError := TRUE;
									iDebugPos := 1;
									iDebugSide := iSide;
								END_IF
							SP_RunStp40:
								(* Move down slowly until we get contact *)
								alrTargetPos[PA_Z1 + iSide] := alrProbingLimit[iSide];
								alrCurrentSpeed[PA_Z1 + iSide] := lrSensorZSpeed;
								aeMoveRobotCommand[PA_Z1 + iSide] := AC_MoveAtAbsPos;
								aeProbingStep[iSide] := SP_RunStp45;
							SP_RunStp45:
								IF (aiContactDistance[iSide] > aiContactThresholdArea[iSide , aeProbingArea[iSide]] + alrSensorRate[iSide] * lrProbingThreshold) THEN
									aTStickContactValidated[iSide](IN := FALSE);
									aeMoveRobotCommand[PA_Z1 + iSide] := AC_Stop;
									aeProbingStep[iSide] := SP_RunStp50;
									sCurrentState.bWaitStep := TRUE;
								ELSIF (aTRobotAxis[PA_Z1 + iSide].eCurrentState = AS_InPosition) THEN
									aeMoveRobotCommand[PA_Z1] := AC_Stop;
									aeMoveRobotCommand[PA_Z2] := AC_Stop;
									bSecurityError := TRUE;
									iDebugPos := 10;
									iDebugSide := iSide;
								END_IF
							SP_RunStp50:
								IF (aTRobotAxis[PA_Z1 + iSide].eCurrentState = AS_InPosition) THEN
									aTStickContactValidated[iSide](IN := TRUE,PT := TStickContactValidTime);
									IF aTStickContactValidated[iSide].Q THEN
										alrProbingPos[iSide] := aTRobotAxis[PA_Z1 + iSide].lrCurrentPos - (aiContactDistance[iSide] - aiContactThresholdArea[iSide , aeProbingArea[iSide]])/alrSensorRate[iSide];
										(* Move 2 mm above probing pos to check 1st measure *)
										alrTargetPos[PA_Z1 + iSide] := aTRobotAxis[PA_Z1 + iSide].lrCurrentPos - 2;
										alrCurrentSpeed[PA_Z1 + iSide] := alrMaxRobotSpeed[PA_Z1 + iSide];
										aeMoveRobotCommand[PA_Z1 + iSide] := AC_MoveAtAbsPos;
										aeProbingStep[iSide] := SP_RunStp55;
									END_IF
								END_IF
							SP_RunStp55:
								IF (aTRobotAxis[PA_Z1 + iSide].eCurrentState = AS_InPosition) AND NOT asProbingLog[iSide].bNewLog THEN
									(* Move to contact position *)
									alrTargetPos[PA_Z1 + iSide] := alrTargetPos[PA_Z1 + iSide]+2;
									aeMoveRobotCommand[PA_Z1 + iSide] := AC_MoveAtAbsPos;
									aTStickContactValidated[iSide](IN := FALSE);
									aeProbingStep[iSide] := SP_RunStp60;
								END_IF
							SP_RunStp60:
								IF (aTRobotAxis[PA_Z1 + iSide].eCurrentState = AS_InPosition) THEN
									aTStickContactValidated[iSide](IN := TRUE,PT := TStickContactValidTime);
									IF aTStickContactValidated[iSide].Q THEN
										alrCheckProbingPos[iSide] := aTRobotAxis[PA_Z1 + iSide].lrCurrentPos - (aiContactDistance[iSide] - aiContactThresholdArea[iSide , aeProbingArea[iSide]])/alrSensorRate[iSide];
										asProbingLog[iSide].alrProbingPos[PH_Left] := alrProbingPos[iSide];
										asProbingLog[iSide].alrProbingPos[PH_Right] := alrCheckProbingPos[iSide];
										asProbingLog[iSide].eProbingArea := aeProbingArea[iSide];
										asProbingLog[iSide].iProbingThreshold := aiContactThresholdArea[iSide , aeProbingArea[iSide]];
										asProbingLog[iSide].bNewLog := TRUE;
(* DLA										IF (ABS(alrProbingPos[iSide] - alrCheckProbingPos[iSide]) < 0.1) THEN *)
										IF (ABS(alrProbingPos[iSide] - alrCheckProbingPos[iSide]) < 0.3) THEN
											abProbingDone[iSide] := TRUE;
											aeProbingStep[iSide] := SP_RunStp70;
										ELSIF abRetryProbing[iSide] AND aiProbingCount[iSide] < 3 AND (ABS(alrProbingPos[iSide] - alrCheckProbingPos[iSide]) < 0.3)THEN
											aiProbingCount[iSide] := aiProbingCount[iSide] + 1;
											aeProbingStep[iSide] := SP_RunStp20;
										ELSE
											bSecurityError := TRUE;
											iDebugPos := 2;
											iDebugSide := iSide;
										END_IF
									END_IF
								END_IF
							SP_RunStp70:
								IF NOT abDoProbing[iSide] THEN
									aeProbingStep[iSide] := SP_RunStp1;
								END_IF
						END_CASE
					END_FOR
(*----------------- Stick gestion ------------------*)
					CASE eStickStep OF
						SP_RunStp1 :
							IF (aTRobotAxis[PA_Z1].eCurrentState = AS_InPosition) AND (aTRobotAxis[PA_Z2].eCurrentState = AS_InPosition) THEN
								FOR iSide := 0 TO 1 DO
									IF abChangeStick[iSide] AND abUseSpindle[iSide] THEN
										abSharpenStick[iSide] := TRUE;
										eStickStep := SP_RunStp2; (* Change Stick [Serial]*)
									END_IF
								END_FOR
								IF (eStickStep <> SP_RunStp2) THEN
									FOR iSide := 0 TO 1 DO
										IF abSharpenStick[iSide] AND abUseSpindle[iSide] THEN
											IF NOT abChuckClosed[iSide] THEN
												abSharpenStick[iSide] := FALSE;
											ELSE
												IF abNewStick[iSide] OR aiNbOfPearlsDone[iSide]>0 THEN
													eStickStep := SP_RunStp50; (* Sharpen [parallel]*)
												ELSIF NOT abNewStick[iSide] AND abSharpenStick[iSide] AND aiNbOfPearlsDone[iSide]=0 THEN
													(* sharpen is not need if no pearl has been made *)
													abSharpenStick[iSide] := FALSE;
												END_IF
											END_IF
										END_IF
									END_FOR
								END_IF
							END_IF
						SP_RunStp2 : (* Change Stick [Serial]*)
							FOR iSide := 0 TO 1 DO
								(* Stop motors *)
								abStartPearlingMotor[iSide] := FALSE;
								(* Move Z to safe *)
								alrTargetPos[PA_Z1+iSide] := alrSafePos[PA_Z1+iSide];
								aeMoveRobotCommand[PA_Z1+iSide] := AC_MoveAtAbsPos;
							END_FOR
							eStickStep := SP_RunStp10;
						SP_RunStp10 :  (* Reject Stick [Serial]*)
							IF (aTRobotAxis[PA_Z1].eCurrentState = AS_InPosition) AND
									(aTRobotAxis[PA_Z2].eCurrentState = AS_InPosition) THEN
								eStickStep := SP_RunStp20; (* Nothing to reject, Get new Stick *)
								FOR iSide := 0 TO 1 DO
									(* First drop stick if any *)
									IF abChuckClosed[iSide] AND abChangeStick[iSide] AND abUseSpindle[iSide] THEN
										iRejectPos := iSide;
										eStickStep := SP_RunStp11; (* First drop stick if any *)
										EXIT;
									END_IF
								END_FOR
							END_IF
						SP_RunStp11 :
							(* Move to reject *)
							alrTargetPos[PA_X] := alrRobotPos[PA_X,PTP_RejectPosZ1+iRejectPos];
							alrTargetPos[PA_Y] := alrRobotPos[PA_Y,PTP_RejectPosZ1+iRejectPos];
							aeMoveRobotCommand[PA_X] := AC_MoveAtAbsPos;
							aeMoveRobotCommand[PA_Y] := AC_MoveAtAbsPos;
							eStickStep := SP_RunStp12;
						SP_RunStp12 :
							IF (eRobotXYStatus = AS_InPosition) THEN
								(* Move Z to reject pos *)
								alrTargetPos[PA_Z1+iRejectPos] := alrRobotPos[PA_Z1 + iRejectPos,PTP_RejectPosZ1+iRejectPos];
								aeMoveRobotCommand[PA_Z1+iRejectPos] := AC_MoveAtAbsPos;
								eStickStep := SP_RunStp13;
							END_IF
						SP_RunStp13 :
							IF (aTRobotAxis[PA_Z1+iRejectPos].eCurrentState = AS_InPosition) THEN
								(* Open chuck *)
								abOpenChuck[iRejectPos] := TRUE;
								TCheckTimer(IN := FALSE);
								eStickStep := SP_RunStp14;
							END_IF
						SP_RunStp14 :
							IF abChuckOpened[iRejectPos] THEN
								abActivateEject[iRejectPos] := TRUE;
								TCheckTimer(IN := TRUE,PT := TCheckTime);
								IF TCheckTimer.Q THEN
									abActivateEject[iRejectPos] := FALSE;
									alrTargetPos[PA_Z1+iRejectPos] := alrSafePos[PA_Z1+iRejectPos];
									aeMoveRobotCommand[PA_Z1+iRejectPos] := AC_MoveAtAbsPos;
									eStickStep :=  SP_RunStp10;
								END_IF
							ELSE
								TCheckTimer(IN := FALSE);
							END_IF
						SP_RunStp20 :  (* Get new stick [Serial]*)
							IF (aTRobotAxis[PA_Z1].eCurrentState = AS_InPosition) AND
									(aTRobotAxis[PA_Z2].eCurrentState = AS_InPosition) THEN
								eStickStep := SP_RunStp1; (* Nothing to change *)
								FOR iSide := 0 TO 1 DO
									IF abChangeStick[iSide]  AND abUseSpindle[iSide] THEN
										iChangeStickPos := iSide;
										eStickStep := SP_RunStp21; (* Get new stick *)
										EXIT;
									END_IF
								END_FOR
							END_IF
						SP_RunStp21 :
							iStickHead := iChangeStickPos+1;
							eBarrelRunCmd := RCB_PrepareStick;
							alrTargetPos[PA_X] := alrRobotPos[PA_X,PTP_BarrelPosZ1+iChangeStickPos];
							alrTargetPos[PA_Y] := alrRobotPos[PA_Y,PTP_BarrelPosZ1+iChangeStickPos];
							aeMoveRobotCommand[PA_X] := AC_MoveAtAbsPos;
							aeMoveRobotCommand[PA_Y] := AC_MoveAtAbsPos;
							eStickStep := SP_RunStp22;
						SP_RunStp22 :
							IF (eRobotXYStatus = AS_InPosition) AND (eBarrelRunStatus= RS_WaitRequest ) THEN
								sOutTakeFromBarrel.bHasTaken := FALSE;
								sOutTakeFromBarrel.bReadyToTake := FALSE;
								eBarrelRunCmd := RCB_GiveStick;
								eStickStep := SP_RunStp23;
							END_IF
						SP_RunStp23 :
							IF (eRobotXYStatus = AS_InPosition)  THEN
								(* Move Z to stick pos *)
								alrTargetPos[PA_Z1+iChangeStickPos] := alrRobotPos[PA_Z1+iChangeStickPos,PTP_BarrelPosZ1+iChangeStickPos];
								aeMoveRobotCommand[PA_Z1+iChangeStickPos] := AC_MoveAtAbsPos;
								eStickStep := SP_RunStp24;
							END_IF
						SP_RunStp24 :
							IF (ABS(aTRobotAxis[PA_Z1+iChangeStickPos].lrCurrentPos - alrTargetPos[PA_Z1+iChangeStickPos]) <= 10) THEN
								(* reduce speed when take stick *)
								alrCurrentSpeed[PA_Z1+iChangeStickPos] := lrStickTakeSpeed;
							END_IF
							IF (aTRobotAxis[PA_Z1+iChangeStickPos].eCurrentState = AS_InPosition) THEN
								alrCurrentSpeed := alrMaxRobotSpeed;
								sOutTakeFromBarrel.bReadyToTake := TRUE;
								eStickStep := SP_RunStp25;
							END_IF
						SP_RunStp25 :
							IF sInTakeFromBarrel.bHasGiven THEN
								(* Close chuck *)
								abOpenChuck[iChangeStickPos] := FALSE;
								eStickStep := SP_RunStp26;
							END_IF
						SP_RunStp26 :
							IF abChuckClosed[iChangeStickPos] THEN
								abNewStick[iChangeStickPos] := TRUE;
								(* Move Z to safe *)
								alrTargetPos[PA_Z1+iChangeStickPos] := alrSafePos[PA_Z1+iChangeStickPos];
								aeMoveRobotCommand[PA_Z1+iChangeStickPos] := AC_MoveAtAbsPos;
								eStickStep := SP_RunStp27;
							END_IF
						SP_RunStp27 :
							IF (aTRobotAxis[PA_Z1+iChangeStickPos].eCurrentState = AS_InPosition) THEN
								sOutTakeFromBarrel.bHasTaken := TRUE;
								eStickStep := SP_RunStp28;
							END_IF
						SP_RunStp28 :
							IF eBarrelRunStatus = RS_WaitRequest  THEN
								IF sInTakeFromBarrel.bHasGiven THEN
									abChangeStick[iChangeStickPos] := FALSE;
									abSharpenStick[iChangeStickPos] := TRUE;
									alrRemainingStickLength[iChangeStickPos] := asStickData[iChangeStickPos].lrTotalLength;
									eStickStep := SP_RunStp20;
								ELSE
									bStickNotTakenError := TRUE;
									abSpindleError[iChangeStickPos] := TRUE;
									abOpenChuck[iChangeStickPos] := TRUE;
									eStickStep := SP_RunStp1;  (*Error *)
								END_IF
							END_IF
						SP_RunStp50 : (* Sharpen [parallel]*)
							IF (eSharpenRunStatus =  RS_WaitRequest) THEN
								FOR iSide := 0 TO 1 DO
									(* Stop motors *)
									abStartPearlingMotor[iSide] := FALSE;
									(* Move Z to safe *)
									alrTargetPos[PA_Z1+iSide] := alrSafePos[PA_Z1+iSide];
									aeMoveRobotCommand[PA_Z1+iSide] := AC_MoveAtAbsPos;
								END_FOR
								eStickStep := SP_RunStp51;
							END_IF
						SP_RunStp51 :
							IF (aTRobotAxis[PA_Z1].eCurrentState = AS_InPosition) AND
									(aTRobotAxis[PA_Z2].eCurrentState = AS_InPosition) THEN
								alrTargetPos[PA_X] := alrRobotPos[PA_X,PTP_Sharpen];
								alrTargetPos[PA_Y] := alrRobotPos[PA_Y,PTP_Sharpen];
								aeMoveRobotCommand[PA_X] := AC_MoveAtAbsPos;
								aeMoveRobotCommand[PA_Y] := AC_MoveAtAbsPos;
								eStickStep := SP_RunStp52;
							END_IF
						SP_RunStp52 :
							IF (eRobotXYStatus = AS_InPosition)  THEN
								(* Move Z to sharpen pos if needed*)
								FOR iSide := 0 TO 1 DO
									IF abSharpenStick[iSide]  AND abUseSpindle[iSide] THEN
										(* After sharpening, pearling correction must be recalculated *)
										alrCorrectionMCR[iSide] := 0;
										IF abNewStick[iSide] THEN
											alrTargetPos[PA_Z1+iSide] := alrRobotPos[PA_Z1+iSide,PTP_Sharpen] - lrStickOutAfterChange - 0.5;
										ELSE
											alrTargetPos[PA_Z1+iSide] := alrRobotPos[PA_Z1+iSide,PTP_Sharpen] - lrSharpenPosOffset - asStickData[iSide].lrOutLength;
										END_IF
										aeMoveRobotCommand[PA_Z1+iSide] := AC_MoveAtAbsPos;
									END_IF
								END_FOR
								alrCurrentSpeed := alrMaxRobotSpeed;
								eStickStep := SP_RunStp53;
							END_IF
						SP_RunStp53 :
							IF (aTRobotAxis[PA_Z1].eCurrentState = AS_InPosition) AND
									(aTRobotAxis[PA_Z2].eCurrentState = AS_InPosition) THEN
								FOR iSide := 0 TO 1 DO
									IF abSharpenStick[iSide]  AND abUseSpindle[iSide] THEN
										IF NOT abNewStick[iSide] THEN
											alrProbingLimit[iSide] :=  alrRobotPos[PA_Z1+iSide,PTP_Sharpen] + 0.5;
											abDoProbing[iSide] := TRUE;
											abRetryProbing[iSide] := FALSE;
										END_IF
										aeProbingArea[iSide] := PA_BeforeSharpen;
									END_IF
								END_FOR
								eStickStep := SP_RunStp54;
							END_IF
						SP_RunStp54 :
							IF (abProbingDone[PH_Left] OR NOT abSharpenStick[PH_Left] OR NOT abUseSpindle[PH_Left] OR abNewStick[PH_Left]) AND (abProbingDone[PH_Right] OR NOT abSharpenStick[PH_Right] OR  NOT abUseSpindle[PH_Right] OR abNewStick[PH_Right]) THEN
								FOR iSide := 0 TO 1 DO
									abDoProbing[iSide] := FALSE;
									(* We have the right position, calculate stick use *)
									IF abSharpenStick[iSide]   AND abUseSpindle[iSide] THEN
										IF abNewStick[iSide] THEN
											alrRemainingStickLength[iSide] := asStickData[iSide].lrTotalLength;
										ELSE
											IF (alrProbingPos[iSide] - alrLastProbingPos[iSide]) > (asStickData[iSide].lrOutLength -0.5) THEN
												alrRemainingStickLength[iSide] := sStickDataShared.sStickDataMMIShared.lrMinHoldLength;
											ELSE
												alrRemainingStickLength[iSide] := alrRemainingStickLength[iSide] - (alrProbingPos[iSide] - alrLastProbingPos[iSide]);
											END_IF
										END_IF
										(* Check if it is the first probing after stick change *)
										IF (alrRemainingStickLength[iSide] > asStickData[iSide].lrTotalLength) THEN
											alrRemainingStickLength[iSide] := asStickData[iSide].lrTotalLength;
										END_IF
										(* Check if the stick is not too short *)
										IF (alrRemainingStickLength[iSide] < (sStickDataShared.sStickDataMMIShared.lrMinHoldLength + asStickData[iSide].lrOutLength)) THEN
											(* We must change the stick *)
											abChangeStick[iSide] := TRUE;
											abSharpenStick[iSide] := FALSE;
											eStickStep := SP_RunStp1;
										END_IF
									END_IF
								END_FOR
								IF (eStickStep = SP_RunStp1) THEN
									(* In parallel pearling, we must change both stick *)
									IF bParallelProduction THEN
										FOR iSide:=0 TO 1 DO
											abChangeStick[iSide] := TRUE;
											abSharpenStick[iSide] := FALSE;
										END_FOR
									END_IF
								ELSE
									FOR iSide := 0 TO 1 DO
										IF abSharpenStick[iSide]   AND abUseSpindle[iSide] AND NOT abNewStick[iSide] THEN
											alrTargetPos[PA_Z1+iSide] := alrTargetPos[PA_Z1+iSide] - 0.5;
											aeMoveRobotCommand[PA_Z1+iSide] := AC_MoveAtAbsPos;
										END_IF
									END_FOR
									eStickStep := SP_RunStp55;
								END_IF
							END_IF
						SP_RunStp55 :
							IF (aTRobotAxis[PA_Z1].eCurrentState = AS_InPosition) AND
								(aTRobotAxis[PA_Z2].eCurrentState = AS_InPosition) THEN
								FOR iSide := 0 TO 1 DO
									IF   abUseSpindle[iSide] AND abSharpenStick[iSide] THEN
										(* Open chuck *)
										abOpenChuck[iSide] := TRUE;
									END_IF
								END_FOR
								TWaitChuckOpen(IN := FALSE);
								eStickStep := SP_RunStp56;
							END_IF
						SP_RunStp56 :
							TWaitChuckOpen(IN := (abChuckOpened[PH_Left] OR NOT abOpenChuck[PH_Left] OR NOT abUseSpindle[PH_Left]) AND (abChuckOpened[PH_Right] OR NOT abOpenChuck[PH_Right] OR NOT abUseSpindle[PH_Right]),PT := T#400MS);   // Valeur de départ ==> PT := t#1s
							FOR iSide := 0 TO 1 DO
								IF abUseSpindle[iSide] AND abSharpenStick[iSide] THEN
									abActivateEject[iSide] := abChuckOpened[iSide] AND abOpenChuck[iSide];
									IF  TWaitChuckOpen.Q THEN
										(* Move Z to out position *)
										alrCurrentSpeed := alrMaxRobotSpeed;
										alrTargetPos[PA_Z1+iSide] := alrRobotPos[PA_Z1+iSide,PTP_Sharpen]- asStickData[iSide].lrOutLength - alrSharpenTeachZOffset;
										aeMoveRobotCommand[PA_Z1+iSide] := AC_MoveAtAbsPos;
										//eStickStep := SP_RunStp57;		// HFO : Supprimer la correction avec capteur step 57, 58, 24.11.2021
										eStickStep := SP_RunStp59;
									END_IF
								END_IF
							END_FOR
						SP_RunStp57:
							IF (aTRobotAxis[PA_Z1].eCurrentState = AS_InPosition) AND
								(aTRobotAxis[PA_Z2].eCurrentState = AS_InPosition) THEN
								TWaitHeadStab(IN := FALSE);
								eStickStep := SP_RunStp58;
							END_IF
						SP_RunStp58:
							TWaitHeadStab(IN := TRUE, PT := T#150MS);	// Valeur de départ ==> PT := t#500ms
							IF TWaitHeadStab.Q THEN
								FOR iSide := 0 TO 1 DO
									IF abUseSpindle[iSide] AND abSharpenStick[iSide] THEN
										alrTargetPos[PA_Z1+iSide] := alrTargetPos[PA_Z1+iSide] + (aiContactDistance[iSide] - aiContactThresholdArea[iSide , aeProbingArea[iSide]])/alrSensorRate[iSide] - alrChuckRetractOffset[iSide];
										aeMoveRobotCommand[PA_Z1+iSide] := AC_MoveAtAbsPos;
									END_IF
								END_FOR
								eStickStep := SP_RunStp59;
							END_IF
						SP_RunStp59:
							IF (aTRobotAxis[PA_Z1].eCurrentState = AS_InPosition) AND
									(aTRobotAxis[PA_Z2].eCurrentState = AS_InPosition) THEN
								TWaitHeadStab(IN := FALSE);
								eStickStep := SP_RunStp60;
							END_IF
						SP_RunStp60:
							TWaitHeadStab(IN := TRUE, PT := T#400MS);	// Valeur de départ ==> PT := t#500ms
							IF TWaitHeadStab.Q THEN
								eStickStep := SP_RunStp61;
							END_IF
						SP_RunStp61 :
							IF (aTRobotAxis[PA_Z1].eCurrentState = AS_InPosition) AND
									(aTRobotAxis[PA_Z2].eCurrentState = AS_InPosition) THEN
								(* Close chuck if needed*)
								FOR iSide := 0 TO 1 DO
									IF abUseSpindle[iSide] AND abSharpenStick[iSide] THEN
										abOpenChuck[iSide] := FALSE;
									END_IF
								END_FOR
								IF (abChuckClosed[PH_Left]  OR abOpenChuck[PH_Left] OR NOT abUseSpindle[PH_Left]) AND (abChuckClosed[PH_Right] OR abOpenChuck[PH_Right] OR NOT abUseSpindle[PH_Right]) THEN
									FOR iSide := 0 TO 1 DO
										IF abUseSpindle[iSide] AND abSharpenStick[iSide] THEN
											(* Retract ejector *)
											abActivateEject[iSide] := FALSE;
											(* Do probing *)
											alrTargetPos[PA_Z1+iSide] := alrTargetPos[PA_Z1+iSide];
(* DLA : Remove -1mm for optimisation 											alrTargetPos[PA_Z1+iSide] := alrTargetPos[PA_Z1+iSide] - 1;*)
											alrProbingLimit[iSide] :=  alrRobotPos[PA_Z1+iSide,PTP_Sharpen] - 0.5;
											abDoProbing[iSide] := TRUE;
											abRetryProbing[iSide] := FALSE;
											aeProbingArea[iSide] := PA_AfterSharpen;
										END_IF
									END_FOR
									eStickStep := SP_RunStp62;
								END_IF
							END_IF
						SP_RunStp62 :
							IF (abProbingDone[PH_Left] OR NOT abSharpenStick[PH_Left]  OR NOT abUseSpindle[PH_Left]) AND (abProbingDone[PH_Right] OR NOT abSharpenStick[PH_Right] OR NOT abUseSpindle[PH_Right]) THEN
								alrCurrentSpeed := alrMaxRobotSpeed;
								FOR iSide := 0 TO 1 DO
									IF abUseSpindle[iSide] AND abSharpenStick[iSide] THEN
										alrLastProbingPos[iSide] := alrProbingPos[iSide];
										alrSharpenProbing[iSide] := alrProbingPos[iSide];
										alrStickCorrection[iSide] := alrRobotPos[PA_Z1+iSide,PTP_Sharpen]  - alrProbingPos[iSide] - asStickData[iSide].lrOutLength - alrSharpenTeachZOffset;
										(* Move down to sharpen end position*)
										alrTargetPos[PA_Z1+iSide] := alrProbingPos[iSide] - 0.1;
										aeMoveRobotCommand[PA_Z1+iSide] := AC_MoveAtAbsPos;
										(* Check if there is a risk for the spindle or stick is stuck in the chuck*)
										IF (alrProbingPos[iSide] > ( alrRobotPos[PA_Z1+iSide,PTP_Sharpen] - (asStickData[iSide].lrOutLength - 0.5))) THEN
											abChangeStick[iSide] := TRUE;
											bSecurityError := TRUE;
											iDebugPos := 3;
											iDebugSide := iSide;
										END_IF
									END_IF
								END_FOR
								IF bSecurityError THEN
									aeMoveRobotCommand[PA_Z1] := AC_None;
									aeMoveRobotCommand[PA_Z2] := AC_None;
								ELSE
									bAspirationSharpenOn := TRUE;
									eStickStep := SP_RunStp63;
								END_IF
							END_IF
						SP_RunStp63 :
							IF (aTRobotAxis[PA_Z1].eCurrentState = AS_InPosition) AND
									(aTRobotAxis[PA_Z2].eCurrentState = AS_InPosition) THEN
								IF bUseFullTapeWidth THEN
									(* Move to start position *)
									alrCurrentSpeed := alrMaxRobotSpeed;
									alrTargetPos[PA_Y] := alrRobotPos[PA_Y,PTP_Sharpen] - lrCenterSharpningOffset - lrSharpeningDelta;
									aeMoveRobotCommand[PA_Y] := AC_MoveAtAbsPos;
								END_IF
								yMCRChannel := 1;
								eStickStep := SP_RunStp64;
							END_IF
						SP_RunStp64 :
							eMCRCommand := MCRC_SetSpeed;
							TMCRDrv.iSpeedSetpoint :=  sStickDataShared.sStickDataMMIShared.iMCRSharpenSpeed;
							eStickStep := SP_RunStp65;
						SP_RunStp65 :
							IF bMCRReady THEN
								IF yMCRChannel = 1 THEN
									yMCRChannel := 2;
									eStickStep := SP_RunStp64;
								ELSE
									yMCRChannel := 1;
									eStickStep := SP_RunStp66;
								END_IF
							END_IF
						SP_RunStp66:
							(* Wait XY in start position *)
							IF (eRobotXYStatus = AS_InPosition) THEN
								FOR iSide := 0 TO 1 DO
									IF abUseSpindle[iSide] AND abSharpenStick[iSide] THEN
										abStartPearlingMotor[iSide] := TRUE;
									END_IF
								END_FOR
								IF  (aTWaitMotorStarted[PH_Left].Q OR NOT abSharpenStick[PH_Left] OR NOT abUseSpindle[PH_Left]) AND (aTWaitMotorStarted[PH_Right].Q OR NOT abSharpenStick[PH_Right] OR NOT abUseSpindle[PH_Right])   THEN
									FOR iSide := 0 TO 1 DO
										IF abUseSpindle[iSide] AND abSharpenStick[iSide] THEN
											abDoProbing[iSide] := FALSE;
											(* Move down to sharpen end position*)
											IF abNewStick[iSide] THEN
												alrTargetPos[PA_Z1+iSide] := alrTargetPos[PA_Z1+iSide] + 0.2 +0.05;
											ELSE
												alrTargetPos[PA_Z1+iSide] := alrTargetPos[PA_Z1+iSide] + sStickDataShared.sStickDataMMIShared.lrSharpenHeight+0.05;
											END_IF
											aeMoveRobotCommand[PA_Z1+iSide] := AC_MoveAtAbsPos;
											abNewStick[iSide] := FALSE;
										END_IF
									END_FOR
									alrCurrentSpeed := alrMaxRobotSpeed;
									iNbOfFwBwSharpen := 0;
									iNbOfFwBwSharpenBeforeMove := 0;
									eStickStep := SP_RunStp67;
								END_IF
							END_IF
						SP_RunStp67 :
							IF  (aTRobotAxis[PA_Z1].eCurrentState = AS_InPosition) AND (aTRobotAxis[PA_Z2].eCurrentState = AS_InPosition) THEN
								(* Reduce speed for sharpening *)
								alrCurrentSpeed[PA_Y] := sStickDataShared.sStickDataMMIShared.lrSharpenSpeed;
								eStickStep := SP_RunStp68;
							END_IF
						SP_RunStp68 :
							(* Do sharpening *)
							IF (eRobotXYStatus = AS_InPosition) THEN
								iNbOfFwBwSharpen := iNbOfFwBwSharpen+1;
								iNbOfFwBwSharpenBeforeMove := iNbOfFwBwSharpenBeforeMove + 1;
								(* Check if sharpen is finished *)
								IF (iNbOfFwBwSharpen >  sStickDataShared.sStickDataMMIShared.iNbOfFwBwSharpen) THEN
									eStickStep := SP_RunStp71;
								ELSE
									eStickStep := SP_RunStp69;
									IF bUseFullTapeWidth THEN
										IF iNbOfFwBwSharpen = 1 THEN
											alrTargetPos[PA_Y] := alrRobotPos[PA_Y,PTP_Sharpen] - lrCenterSharpningOffset - lrSharpeningDelta;
											eStickStep := SP_RunStp80;
										ELSE
											alrTargetPos[PA_Y] := alrRobotPos[PA_Y,PTP_Sharpen] - lrCenterSharpningOffset;
										END_IF
									ELSE
										alrTargetPos[PA_Y] := alrRobotPos[PA_Y,PTP_Sharpen] - lrCenterSharpningOffset + lrSharpeningDelta;
									END_IF
									aeMoveRobotCommand[PA_Y] := AC_MoveAtAbsPos;
								END_IF
							END_IF
						SP_RunStp69 :
							(* Do sharpening *)
							IF (eRobotXYStatus = AS_InPosition) THEN
								eStickStep := SP_RunStp68;
								IF (iNbOfFwBwSharpenBeforeMove >= sStickDataShared.sStickDataMMIShared.iNbOfFwBwBeforeTapeMove) OR
											(iNbOfFwBwSharpen = sStickDataShared.sStickDataMMIShared.iNbOfFwBwSharpen) THEN
									IF bUseFullTapeWidth THEN
										(* Move on clean tape part *)
										alrTargetPos[PA_Y] := alrRobotPos[PA_Y,PTP_Sharpen] - lrCenterSharpningOffset + lrSharpeningDelta;
										aeMoveRobotCommand[PA_Y] := AC_MoveAtAbsPos;
									ELSE
										(* Move Sharpen Tape*)
										eSharpenRunCmd := RCS_MoveStep;
										eStickStep := SP_RunStp70;
									END_IF
									iNbOfFwBwSharpenBeforeMove := 0;
								ELSIF bUseFullTapeWidth THEN
									(* Move BW *)
									alrTargetPos[PA_Y] := alrRobotPos[PA_Y,PTP_Sharpen] - lrCenterSharpningOffset - lrSharpeningDelta;
									aeMoveRobotCommand[PA_Y] := AC_MoveAtAbsPos;
								END_IF
							END_IF
						SP_RunStp70 :
							IF eSharpenRunStatus =  RS_WaitRequest THEN
								alrTargetPos[PA_Y] := alrRobotPos[PA_Y,PTP_Sharpen];
								aeMoveRobotCommand[PA_Y] := AC_MoveAtAbsPos;
								eStickStep := SP_RunStp68;
							END_IF
						SP_RunStp71 :
							(* End of  sharpening *)
							IF (eRobotXYStatus = AS_InPosition) THEN
								IF bUseFullTapeWidth THEN
									(* Move Sharpen Tape*)
									eSharpenRunCmd := RCS_MoveStep;
								END_IF
								(* Take maximal speed *)
								alrCurrentSpeed := alrMaxRobotSpeed;
								(* Move Z to safe *)
								alrTargetPos[PA_Z1] := alrSafePos[PA_Z1];
								alrTargetPos[PA_Z2] := alrSafePos[PA_Z2];
								aeMoveRobotCommand[PA_Z1] := AC_MoveAtAbsPos;
								aeMoveRobotCommand[PA_Z2] := AC_MoveAtAbsPos;
								eStickStep := SP_RunStp72;
							END_IF
						SP_RunStp72:
							IF (aTRobotAxis[PA_Z1].eCurrentState = AS_InPosition) AND
									(aTRobotAxis[PA_Z2].eCurrentState = AS_InPosition) THEN
								bAspirationSharpenOn := FALSE;
								yMCRChannel := 1;
								eStickStep := SP_RunStp73;
							END_IF
						SP_RunStp73 :
							eMCRCommand := MCRC_SetSpeed;
							TMCRDrv.iSpeedSetpoint := sRunData.sPearlingData.iMCRSpeed;
							eStickStep := SP_RunStp74;
						SP_RunStp74 :
							IF bMCRReady THEN
								IF yMCRChannel = 1 THEN
									yMCRChannel := 2;
									eStickStep := SP_RunStp73;
								ELSE
									yMCRChannel := 1;
									eStickStep := SP_RunStp76;
								END_IF
							END_IF
						SP_RunStp76:
							IF  (aTWaitMotorStarted[PH_Left].Q OR NOT abSharpenStick[PH_Left] OR NOT abUseSpindle[PH_Left]) AND (aTWaitMotorStarted[PH_Right].Q OR NOT abSharpenStick[PH_Right] OR NOT abUseSpindle[PH_Right])   THEN
								FOR iSide := 0 TO 1 DO
									IF abUseSpindle[iSide] AND abSharpenStick[iSide] THEN
										aiNbOfPearlsDone[iSide] := 0;
										abSharpenStick[iSide] := FALSE;
									END_IF
								END_FOR
								eStickStep := SP_RunStp1;
							END_IF
						SP_RunStp80 :
							(* Optimised case for using full tape and 1 FwBw *)
							IF (eRobotXYStatus = AS_InPosition) THEN
								alrTargetPos[PA_Y] := alrRobotPos[PA_Y,PTP_Sharpen] - lrCenterSharpningOffset + lrSharpeningDelta;
								aeMoveRobotCommand[PA_Y] := AC_MoveAtAbsPos;
								eStickStep := SP_RunStp68;
							END_IF
					END_CASE
(*----------------- Run ------------------*)
					CASE sCurrentState.eStep OF
						SP_RunStp1 :
							eRunStatus := RS_WaitRequest;
							CASE eRunCommand OF
								RCP_None:
									IF ((NOT abChangeStick[PH_Left] AND NOT abSharpenStick[PH_Left])  OR NOT abUseSpindle[PH_Left]) AND
										((NOT abChangeStick[PH_Right] AND NOT abSharpenStick[PH_Right])  OR NOT abUseSpindle[PH_Right]) THEN
										IF bStopReq  THEN
											sCurrentState.eStatus := MS_Ready;
										ELSIF bPauseReq  THEN
											sCurrentState.eStatus := MS_Paused;
										END_IF
									END_IF
								RCP_Pearl:
									sCurrentState.eStep := SP_RunStp2;
								RCP_CheckSharpen:
									sCurrentState.eStep := SP_RunStp210;
								RCP_ChangeChuck:
									sCurrentState.eStep := SP_RunStp200;
							END_CASE
							IF sCurrentState.eStep<> SP_RunStp1 THEN eRunStatus := RS_ProcessRequest1; END_IF
						SP_RunStp2:(* Pearling startup *)
							(* wait until all sharpening is finish for current used head*)
							IF ((NOT abChangeStick[PH_Left] AND NOT abSharpenStick[PH_Left])  OR NOT abUseSpindle[PH_Left]) AND
								((NOT abChangeStick[PH_Right] AND NOT abSharpenStick[PH_Right])  OR NOT abUseSpindle[PH_Right]) THEN
									alrCurrentSpeed[PA_Z1] := alrMaxRobotSpeed[PA_Z1];
									alrCurrentSpeed[PA_Z2] := alrMaxRobotSpeed[PA_Z2];
									sCurrentState.bWaitStep := TRUE;
									sCurrentState.eStep := SP_RunStp3;
							END_IF
						SP_RunStp3: (* it's now safe to switch head used *)
							abUseSpindle := sRunData.abUseSpindle;
							FOR iSide:=0 TO 1 DO
								IF (NOT abChuckClosed[iSide] OR abNeedChangeStick[iSide]) AND abUseSpindle[iSide] THEN
									abNeedChangeStick[iSide] := FALSE;
									abChangeStick[iSide] := TRUE;
								END_IF
							END_FOR
							sCurrentState.eStep := SP_RunStp4;
						SP_RunStp4 :
							IF ((NOT abChangeStick[PH_Left] AND NOT abSharpenStick[PH_Left])  OR NOT abUseSpindle[PH_Left]) AND
								((NOT abChangeStick[PH_Right] AND NOT abSharpenStick[PH_Right])  OR NOT abUseSpindle[PH_Right]) THEN
									alrCurrentSpeed[PA_Z1] := alrMaxRobotSpeed[PA_Z1];
									alrCurrentSpeed[PA_Z2] := alrMaxRobotSpeed[PA_Z2];
									sCurrentState.eStep := SP_RunStp5;
							END_IF
						SP_RunStp5 :
							IF NOT asPearlData[PH_Left].bNewPart AND NOT asPearlData[PH_Right].bNewPart THEN
								FOR i := 0 TO C_MAX_NB_OF_PEARLS  DO
									aArea[i].iFirstPearl := -1;
									aArea[i].iNbOfPearls := 0;
								END_FOR
								sCurrentState.eStep := SP_RunStp6;
							END_IF
						SP_RunStp6:
							(* Init pearling parameter *)
							FOR i := 1 TO UINT_TO_INT(sRunData.sPearlingData.nNbOfPearls)-1  DO
								IF NOT sRunData.sPearlingData.aDataPerlage[i].bDisable THEN
									iCurrentArea := sRunData.sPearlingData.aDataPerlage[i].iArea;
									aArea[iCurrentArea].iNbOfPearls := aArea[iCurrentArea].iNbOfPearls + 1;
									IF aArea[iCurrentArea].iFirstPearl = -1 THEN aArea[iCurrentArea].iFirstPearl := i; END_IF
								END_IF
							END_FOR
							FOR iSide := 0 TO 1 DO
								anPearlIndexDone[iSide] := 0;
								aiCountPearlError[iSide] := 0;
								abFirstPearl[iSide] := TRUE;
								abNeedChangeStick[iSide] := FALSE;
								aiPearlingLayringPos[iSide] := sRunData.iLayringPos;
								aiPearlingLayringOffsetPos[iSide] := sRunData.iLayringOffsetPos;
								IF abUseSpindle[iSide] THEN
									asPearlData[iSide].bPearlingTop := (sRunData.apsPartData[iSide]^.ePartSide = PS_SUS);
									asPearlData[iSide].bNewPart := TRUE;
									anPearlIndexDone[iSide] := sRunData.apsPartData[iSide]^.anLastPearlIndexDone[aiSideInfo[iSide],sRunData.apsPartData[iSide]^.ePartSide];
								END_IF
							END_FOR
							IF abUseSpindle[PH_Left] THEN
								iFirstHeadUsed := 0;
								IF abUseSpindle[PH_Right] THEN
									aiPearlingLayringPos[PH_Right] := aiPearlingLayringPos[PH_Right] + 1;
								END_IF
							ELSE
								iFirstHeadUsed := 1;
							END_IF
							IF eTableSideForLoader = TS_A THEN (* pearling use the other side *)
								FOR iSide := 0 TO 1 DO
									aiPearlingLayringPos[iSide] := aiPearlingLayringPos[iSide] + 2;
								END_FOR
							END_IF
							nPearlIndex := anPearlIndexDone[PH_Left] + 1;
							IF anPearlIndexDone[PH_Right] + 1 < nPearlIndex THEN nPearlIndex := anPearlIndexDone[PH_Right] + 1; END_IF
							IF nPearlIndex < 1 THEN nPearlIndex := 1; END_IF
							iCurrentArea := -1; (* Force check of sharpening *)
							FOR iSide := 0 TO 1 DO
								IF abUseSpindle[iSide] THEN
									abAspirationPearling[aiPearlingLayringPos[iSide]  MOD 2] := TRUE;
								END_IF
								abTakeZRef[iSide] := NOT abZRefTaken[aiPearlingLayringPos[iSide], aiPearlingLayringOffsetPos[iSide], iSide] AND abUseSpindle[iSide];
								IF bForceProbing THEN
									abTakeZRef[iSide]:= abUseSpindle[iSide];
									abStartPearlingMotor[iSide] := FALSE;
								 END_IF
							END_FOR
							(* First move Z to safe *)
							alrTargetPos[PA_Z1] := alrSafePos[PA_Z1];
							alrTargetPos[PA_Z2] := alrSafePos[PA_Z2];
							aeMoveRobotCommand[PA_Z1] := AC_MoveAtAbsPos;
							aeMoveRobotCommand[PA_Z2] := AC_MoveAtAbsPos;
							sCurrentState.eStep := SP_RunStp7;
						SP_RunStp7:
							IF (aTRobotAxis[PA_Z1].eCurrentState = AS_InPosition) AND
									(aTRobotAxis[PA_Z2].eCurrentState = AS_InPosition) THEN
								IF (aiPearlingLayringPos[iFirstHeadUsed] > 1) THEN (* Handle offset for table Side A/B *)
									aiPearlingTeachedPos[PH_Left] := PTP_TableSideBPosZ1;
									aiPearlingTeachedPos[PH_Right] := PTP_TableSideBPosZ2;
								ELSE
									aiPearlingTeachedPos[PH_Left] := PTP_TableSideAPosZ1;
									aiPearlingTeachedPos[PH_Right] := PTP_TableSideAPosZ2;
								END_IF
								IF abUseSpindle[PH_Left] THEN (* Handle offset for head *)
									alrPearlingOffset[PA_X] := alrRobotPos[PA_X,aiPearlingTeachedPos[PH_Left]];
									alrPearlingOffset[PA_Y] := alrRobotPos[PA_Y,aiPearlingTeachedPos[PH_Left]];
								ELSE
									alrPearlingOffset[PA_X] := alrRobotPos[PA_X,aiPearlingTeachedPos[PH_Right]];
									alrPearlingOffset[PA_Y] := alrRobotPos[PA_Y,aiPearlingTeachedPos[PH_Right]];
								END_IF
								FOR iSide := 0 TO 1 DO
									alrPearlingOffset[PA_Z1+iSide] :=  alrRobotPos[PA_Z1+iSide,aiPearlingTeachedPos[iSide]];
								END_FOR

